FUNCTION_BLOCK E_REND_3 (* Rendezvous (AND) of three events (generic FB) *)
  (* Standard: 61499-1 Annex A; Classification: event function block; Function: Rendezvous of three events; Description: Copyright (c) 2017, 2026 fortiss GmbH, HR Agrartechnik GmbH This program and the accompanying materials are made available under the terms of the Eclipse Public License 2.0 which is available at https://www.eclipse.org/legal/epl-2.0/ SPDX-License-Identifier: EPL-2.0 Some portions generated by Gemini CLI *)
  (* Version 1.0, 2026-02-01, Franz Höpfinger, HR Agrartechnik GmbH, Initial creation based on E_REND and E_SPLIT_3 *)
  PACKAGE iec61499::events;
  {SET_ATTRIBUTE(eclipse4diac::core::GenericClassName, 'GEN_E_REND')}
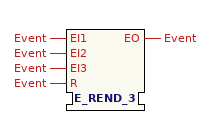
  EVENT_INPUT
    EI1; (* First event to wait for *)
    EI2; (* Second event to wait for *)
    EI3; (* Third event to wait for *)
    R; (* Reset the FB to inital state (i.e., wait again for all events) *)
  END_EVENT
  EVENT_OUTPUT
    EO; (* Triggered when all input events occured at least once *)
  END_EVENT
END_FUNCTION_BLOCK
